FUNCTION_BLOCK FB_SimAxis IMPLEMENTS IAxis
VAR_INPUT
END_VAR
VAR_OUTPUT
END_VAR
VAR
	fActPosition		: LREAL;
	fActVelocity		: LREAL;
	
	bBusy				: BOOL;
	bError				: BOOL;
END_VAR

PROPERTY ActPosition : LREAL
GET
ActPosition := fActPosition;
END_GET
END_PROPERTY

PROPERTY ActVelocity : LREAL
GET
ActVelocity := fActVelocity;
END_GET
END_PROPERTY

PROPERTY Busy : BOOL
GET
Busy := bBusy;
END_GET
END_PROPERTY

METHOD Enable : BOOL
END_METHOD

PROPERTY Enabled : BOOL
GET
END_GET
END_PROPERTY

PROPERTY Error : BOOL
GET
Error := bError;
END_GET
END_PROPERTY

METHOD Execute : BOOL
RETURN;
END_METHOD

METHOD JogFwd : BOOL
VAR_INPUT
	Velocity	: LREAL;
END_VAR
fActVelocity := Velocity;
fActPosition := fActPosition + (Velocity / 101.9);
END_METHOD

METHOD JogRev : BOOL
VAR_INPUT
	Velocity	: LREAL;
END_VAR
fActVelocity := -(Velocity);
fActPosition := fActPosition - (Velocity / 101.9);
END_METHOD

PROPERTY MaxTorque : LREAL
GET
END_GET
SET
END_SET
END_PROPERTY

METHOD MoveAbsolute : BOOL
VAR_INPUT
	(* target position*)
	Target		: LREAL;
	Velocity	: LREAL;
END_VAR
bBusy := TRUE;
IF fActPosition < (Target - 1.5) THEN
	THIS^.JogFwd(Velocity);
	MoveAbsolute := FALSE;
ELSIF fActPosition > (Target + 1.5) THEN
	THIS^.JogRev(Velocity);
	MoveAbsolute := FALSE;
ELSE
	bBusy := FALSE;
	MoveAbsolute := TRUE;
END_IF
END_METHOD

METHOD Reset : BOOL
END_METHOD

METHOD SetHome : BOOL
VAR_INPUT
	Target	: LREAL;
END_VAR
END_METHOD

METHOD StopMove : BOOL
END_METHOD

END_FUNCTION_BLOCK

(* stored: Version 1.1.0.1, ProductVersion 3.1.4024.12
   POU FB_SimAxis: Id {5174d465-34a5-46fe-849e-2e264f751283}, SpecialFunc None
   Property ActPosition: Id {4201ee61-4bae-4420-9906-f329da9b2eaa}
   Get Get: Id {d94d6bf1-7845-4873-9ab0-a9a6000e2001}
   Property ActVelocity: Id {45bf43e1-198c-4715-bb1a-d6a6886e76fc}
   Get Get: Id {cb26f182-28f1-479b-b4b6-c848522e7907}
   Property Busy: Id {795f7e9e-c293-4e15-a769-a5d43da9af34}
   Get Get: Id {c77461da-d17d-46bc-a1c8-c354e196da7d}
   Method Enable: Id {bdc8b238-74ca-4278-ad3a-2a0c80f9cbb6}
   Property Enabled: Id {f3f8d52e-5df6-4243-aa25-918a9e170110}
   Get Get: Id {d88da46b-61c6-47b7-b442-5182c4f2e019}
   Property Error: Id {841c6852-6840-4821-8142-778fe6c0d2aa}
   Get Get: Id {34148eb9-c706-4b25-8997-490489717e3d}
   Method Execute: Id {89a09af4-88ca-434f-b209-f841df8dcc8a}
   Method JogFwd: Id {87e78a3f-8c03-4ed4-8c8a-3309978460dc}
   Method JogRev: Id {dc851cbc-856a-42a3-981c-b3912436c305}
   Property MaxTorque: Id {28351169-0fb5-4ee9-b297-7ac321290eb4}
   Get Get: Id {d9c32682-64c9-405f-9c27-4540ede287fc}
   Set Set: Id {76b8cf73-ae3b-407b-bf89-e40bb50026f9}
   Method MoveAbsolute: Id {25522c8a-7bd7-4697-8c0a-22d3b9a92e61}
   Method Reset: Id {f5a9cd22-7729-4246-9d15-881079fb27b0}
   Method SetHome: Id {9fe7e810-3b40-4c68-944c-d24f373a3e2b}
   Method StopMove: Id {ac02ecb5-302e-4f6e-aacf-d73b1da7ef6a} *)
